INTERFACE I_SessionData EXTENDS I_Disposable

END_INTERFACE

(* stored: Version 1.1.0.1, ProductVersion 3.1.4024.12
   Itf I_SessionData: Id {efd3685a-8f84-4051-baa3-77277d9cbbaa} *)
